FUNCTION_BLOCK Timer
  (* Standard: 61499-2 *)
  (* Version 0.2, 2003-12-04, JHC, Rockwell Automation, Renamed for better indexing. *)
  (* Version 0.1, 2002-11-05, JHC, Rockwell Automation, Corrected missing ST element in Algorithm REQ. *)
  (* Version 0.0, 2000-05-30, JHC, Rockwell Automation *)
  (* Compiler header: package fb.rt.benchmarks.watermonitor; *)
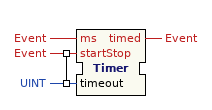
  EVENT_INPUT
    ms; (* millisecond *)
    startStop WITH timeout; (* toggles the timer *)
  END_EVENT
  EVENT_OUTPUT
    timed;
  END_EVENT
  VAR_INPUT
    timeout : UINT := 0; (* timeout value *)
  END_VAR
  VAR
    count : UINT := 0;
  END_VAR
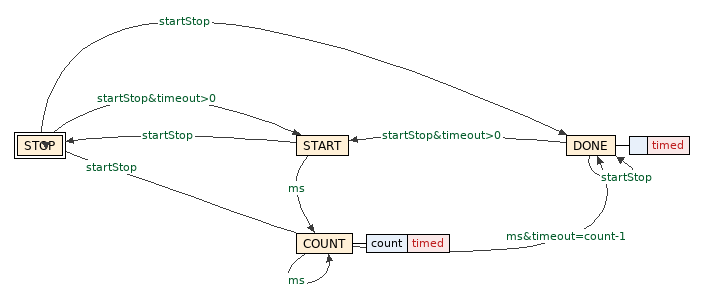
  EC_STATES
    STOP; (* Initial State *)
    START;
    COUNT : count -> timed;
    DONE : -> timed;
  END_STATES
  EC_TRANSITIONS
    STOP TO START := startStop&timeout>0;
    STOP TO DONE := startStop;
    START TO STOP := startStop;
    START TO COUNT := ms;
    COUNT TO STOP := startStop;
    COUNT TO DONE := ms&timeout=count-1;
    COUNT TO COUNT := ms;
    DONE TO START := startStop&timeout>0;
    DONE TO DONE := startStop;
  END_TRANSITIONS
  ALGORITHM count IN ST: (* Initialization algorithm *)
count := count + 1;
  END_ALGORITHM
END_FUNCTION_BLOCK
